INTERFACE I_MoveAbsolute EXTENDS I_StatusEx

PROPERTY Active : BOOL
GET
END_GET
END_PROPERTY

PROPERTY CommandMoveAbsolute : BOOL
SET
END_SET
END_PROPERTY

METHOD MoveAbsolute
VAR_INPUT
    Position	: LREAL;
    Velocity	: LREAL;
    Acceleration	: LREAL := 0.0;
    Deceleration	: LREAL := 0.0;
    Jerk	: LREAL := 0.0;
    BufferMode	: MC_BufferMode := MC_BufferMode.MC_Aborting;
END_VAR
END_METHOD

END_INTERFACE

(* stored: Version 1.1.0.1
   Itf I_MoveAbsolute: Id {7b52c23d-d549-4d14-b715-d0e842580738}
   Property Active: Id {aa5e4d9b-53b9-487d-aa20-131cb555a892}
   Get Get: Id {0e48ad5c-2521-41b7-88a3-39e827f8d022}
   Property CommandMoveAbsolute: Id {8c97d5d2-df79-4b9c-99ac-17d60df5023f}
   Set Set: Id {b3030849-d707-42bf-a5a6-bbde2b420f1c}
   Method MoveAbsolute: Id {6ca50ed1-00a4-4a5f-9fc0-b477fbaad08d} *)
